	                #sFB_TimerOnOffDelay_Hold330(iudi_OnDelayTime := #cudi_PushOutTime,
	                                             ix_SignalToDelay := NOT #sx_LeftExternalRequestHold330
	                                             AND #iqUDT_WorkstationStatus."310".PEC_EoS.PEC
	                                             AND #iqUDT_WorkstationStatus."320".PEC_EoS.PEC
	                                             AND #iqUDT_WorkstationStatus."330".PEC_EoS.PEC,
	                                             ix_Enable := TRUE);

	                #sFB_TimerOnOffDelay_Hold320(iudi_OnDelayTime := #cudi_PushOutTime,
	                                             ix_SignalToDelay := NOT #sx_LeftExternalRequestHold320
	                                             AND #iqUDT_WorkstationStatus."310".PEC_EoS.PEC
	                                             AND #iqUDT_WorkstationStatus."320".PEC_EoS.PEC,
	                                             ix_Enable := TRUE);

	                #sFB_TimerOnOffDelay_Hold310(iudi_OnDelayTime := #cudi_PushOutTime,
	                                             ix_SignalToDelay := NOT #sx_LeftExternalRequestHold310
	                                             AND #iqUDT_WorkstationStatus."310".PEC_EoS.PEC,
	                                             ix_Enable := TRUE);



	            END_REGION

	            REGION 0.4.2 - Delayed start of pushout conveyors after pushout detection
	                #sFB_TimerOnOffDelay_Detect340(iudi_OnDelayTime := #cudi_DetectTime,
	                                               ix_SignalToDelay := NOT #iqUDT_WorkstationStatus."340".PEC_EoS.PEC,
	                                               ix_Enable := TRUE);

	                #sFB_TimerOnOffDelay_Detect330(iudi_OnDelayTime := #cudi_DetectTime,
	                                               ix_SignalToDelay := NOT #iqUDT_WorkstationStatus."330".PEC_EoS.PEC,
	                                               ix_Enable := TRUE);

	                #sFB_TimerOnOffDelay_Detect320(iudi_OnDelayTime := #cudi_DetectTime,
	                                               ix_SignalToDelay := NOT #iqUDT_WorkstationStatus."320".PEC_EoS.PEC,
	                                               ix_Enable := TRUE);

	                #sFB_TimerOnOffDelay_Detect310(iudi_OnDelayTime := #cudi_DetectTime,
	                                               ix_SignalToDelay := NOT #iqUDT_WorkstationStatus."310".PEC_EoS.PEC,
	                                               ix_Enable := TRUE);
	            END_REGION

	            REGION 0.4.3 - Gate conveyor proximity sensor filtered signal

	                #sFB_TimerOnOffDelay_GateIsDown111Filtered(iudi_OnDelayTime := #cudi_GateIsDownFilterTime,
	                                                           iudi_OffDelayTime := 10,
	                                                           ix_SignalToDelay := #ix_GateIsDown111,
	                                                           qx_DelayedSignal => #sx_GateIsDown111Filtered);
	            END_REGION
	        END_REGION

	        REGION 0.5 - Left station activation

	            IF #sx_ActivationLeft
	            THEN
	                #sx_LeftStationActive := TRUE;
	                #iqUDT_LeftWESInterface.PLC2WES.On := TRUE;
	            END_IF;

	            IF #sx_DeactivationLeft
	            THEN
	                #sx_LeftStationActive := FALSE;
	                #iqUDT_LeftWESInterface.PLC2WES.Off := TRUE;
	            END_IF;


	        END_REGION

	    END_IF;

	END_REGION




	REGION 1 - Initial Right station

	    IF #iUDT_Configuration.GlobalConfig.StationVariant = 1 OR #iUDT_Configuration.GlobalConfig.StationVariant = 3 THEN

	        REGION 1.1 - Reset triggers

	            IF #sx_ActivationRight THEN
	                #iqUDT_RightWESInterface.WES2PLC.On := FALSE;
	                #sx_ActivationRight := FALSE;
	            END_IF;

	            IF #sx_DeactivationRight THEN
	                #iqUDT_RightWESInterface.WES2PLC.Off := FALSE;
	                #sx_DeactivationRight := FALSE;
	            END_IF;

	        END_REGION

	        REGION 1.2 - Triggers

	            #sR_TRIG_PEC540(CLK := #iqUDT_WorkstationStatus."540".PEC_EoS.PEC);   //Rising Edge PEC on conveyor 540 for indexing into station count

	            #sR_TRIG_ActivateRightStation(CLK := #iqUDT_RightWESInterface.WES2PLC.On,     //Rising Edge activate right station
	                                          Q => #sx_ActivationRight);

	            #sR_TRIG_DeactivateRightStation(CLK := #iqUDT_RightWESInterface.WES2PLC.Off,   //Rising Edge deactivate right station
	                                            Q => #sx_DeactivationRight);

	        END_REGION

	        REGION 1.3 - Counters

	            REGION 1.3.1 - Count empty stations on right side

	                //If there is no indexing procedure then count empty stations
	                //
	                IF NOT #sx_RightIndexing THEN

	                    #sFB_CountActiveInputs_RightStation(ix_Input1 := #iqUDT_WorkstationStatus."550".PEC_EoS.PEC,
	                                                        ix_Input2 := #iqUDT_WorkstationStatus."560".PEC_EoS.PEC,
	                                                        ix_Input3 := #iqUDT_WorkstationStatus."570".PEC_EoS.PEC,
	                                                        ix_Input4 := #iqUDT_WorkstationStatus."580".PEC_EoS.PEC,
	                                                        ix_Input5 := #iqUDT_WorkstationStatus."590".PEC_EoS.PEC,
	                                                        qi_ActiveInputsCount => #si_RightEmptyStations);
	                END_IF;
	            END_REGION



	            REGION 1.3.2 - Count free spaces on right buffer

	                IF #sx_RightStationActive THEN
	                    #sFB_CountActiveInputs_RightBuffer(ix_Input1 := #iqUDT_WorkstationStatus."520".PEC_EoS.PEC,
	                                                       ix_Input2 := #iqUDT_WorkstationStatus."530".PEC_EoS.PEC,
	                                                       ix_Input3 := #iqUDT_WorkstationStatus."540".PEC_EoS.PEC);
	                ELSE
	                    #sFB_CountActiveInputs_RightBuffer.qi_ActiveInputsCount := 0;
	                END_IF;

	            END_REGION

	        END_REGION

	        REGION 1.4 - Timers

	            REGION 1.4.1 - Right station timers for holding pushout conveyors after pushout

	                #sFB_TimerOnOffDelay_Hold750(iudi_OnDelayTime := #cudi_PushOutTime,
	                                             ix_SignalToDelay := NOT #sx_RightExternalRequestHold750
	                                             AND #iqUDT_WorkstationStatus."710".PEC_EoS.PEC
	                                             AND #iqUDT_WorkstationStatus."720".PEC_EoS.PEC
	                                             AND #iqUDT_WorkstationStatus."730".PEC_EoS.PEC
	                                             AND #iqUDT_WorkstationStatus."740".PEC_EoS.PEC
	                                             AND #iqUDT_WorkstationStatus."750".PEC_EoS.PEC,
	                                             ix_Enable := TRUE);

	                #sFB_TimerOnOffDelay_Hold740(iudi_OnDelayTime := #cudi_PushOutTime,
	                                             ix_SignalToDelay := NOT #sx_RightExternalRequestHold740
	                                             AND #iqUDT_WorkstationStatus."710".PEC_EoS.PEC
	                                             AND #iqUDT_WorkstationStatus."720".PEC_EoS.PEC
	                                             AND #iqUDT_WorkstationStatus."730".PEC_EoS.PEC
	                                             AND #iqUDT_WorkstationStatus."740".PEC_EoS.PEC,
	                                             ix_Enable := TRUE);

	                #sFB_TimerOnOffDelay_Hold730(iudi_OnDelayTime := #cudi_PushOutTime,
	                                             ix_SignalToDelay := NOT #sx_RightExternalRequestHold730
	                                             AND #iqUDT_WorkstationStatus."710".PEC_EoS.PEC
	                                             AND #iqUDT_WorkstationStatus."720".PEC_EoS.PEC
	                                             AND #iqUDT_WorkstationStatus."730".PEC_EoS.PEC,
	                                             ix_Enable := TRUE);

	                #sFB_TimerOnOffDelay_Hold720(iudi_OnDelayTime := #cudi_PushOutTime,
	                                             ix_SignalToDelay := NOT #sx_RightExternalRequestHold720
	                                             AND #iqUDT_WorkstationStatus."710".PEC_EoS.PEC
	                                             AND #iqUDT_WorkstationStatus."720".PEC_EoS.PEC,
	                                             ix_Enable := TRUE);

	                #sFB_TimerOnOffDelay_Hold710(iudi_OnDelayTime := #cudi_PushOutTime,
	                                             ix_SignalToDelay := NOT #sx_RightExternalRequestHold710
	                                             AND #iqUDT_WorkstationStatus."710".PEC_EoS.PEC,
	                                             ix_Enable := TRUE);
	            END_REGION

	            REGION 1.4.2 - Right station delayed start of pushout conveyors

	                #sFB_TimerOnOffDelay_Detect740(iudi_OnDelayTime := #cudi_DetectTime,
	                                               ix_SignalToDelay := NOT #iqUDT_WorkstationStatus."740".PEC_EoS.PEC,
	                                               ix_Enable := TRUE);

	                #sFB_TimerOnOffDelay_Detect730(iudi_OnDelayTime := #cudi_DetectTime,
	                                               ix_SignalToDelay := NOT #iqUDT_WorkstationStatus."730".PEC_EoS.PEC,
	                                               ix_Enable := TRUE);

	                #sFB_TimerOnOffDelay_Detect720(iudi_OnDelayTime := #cudi_DetectTime,
	                                               ix_SignalToDelay := NOT #iqUDT_WorkstationStatus."720".PEC_EoS.PEC,
	                                               ix_Enable := TRUE);

	                #sFB_TimerOnOffDelay_Detect710(iudi_OnDelayTime := #cudi_DetectTime,
	                                               ix_SignalToDelay := NOT #iqUDT_WorkstationStatus."710".PEC_EoS.PEC,
	                                               ix_Enable := TRUE);

	                #sFB_TimerGateTimeout(iudi_OnDelayTime := #cudi_GateTimout,
	                                      ix_SignalToDelay := NOT #sx_GateIsDown111Filtered,
	                                      qx_DelayedSignal => #sx_GateTimeout);

	            END_REGION

	        END_REGION END_IF;

	        REGION 1.5 - Right station activation

	            IF #sx_ActivationRight
	            THEN
	                #sx_RightStationActive := TRUE;
	                #iqUDT_RightWESInterface.PLC2WES.On := TRUE;
	            END_IF;

	            IF #sx_DeactivationRight
	            THEN
	                #sx_RightStationActive := FALSE;
	                #iqUDT_RightWESInterface.PLC2WES.Off := TRUE;
	            END_IF;

	        END_REGION

	    END_IF;

	END_REGION

	REGION 2 - Lift gate

	    IF #iUDT_Configuration.GlobalConfig.StationVariant > 0 THEN

	        // hold gate conveyors after button press if no maintenance is performed
	        IF #sx_GateIsDown111Filtered AND #sR_TRIG_B112.Q AND NOT #sx_MaintenanceIsPerformed THEN
	            #sx_ExternalRequestHoldGate := TRUE;
	            #sx_MaintenanceIsPerformed := TRUE;


	            // release gate conveyors if gate is down maintenance is performed after button press
	        ELSIF #sx_GateIsDown111Filtered AND #sR_TRIG_B111.Q AND #sx_MaintenanceIsPerformed THEN
	            #sx_ExternalRequestHoldGate := FALSE;
	            #sx_MaintenanceIsPerformed := FALSE;

	            // Hold conveyor if there is no maintenance perfomed and gate has been opened
	        ELSIF NOT #sx_GateIsDown111Filtered AND NOT #sx_MaintenanceIsPerformed THEN
	            #sx_ExternalRequestHoldGate := TRUE;
	        END_IF;


	        // Indicate that Gate is down and stopped
	        IF #sx_MaintenanceIsPerformed AND #sx_GateIsDown111Filtered THEN
	            #qx_Light := TRUE;
	            #sx_HornHold := FALSE;

	            //SCADA Signals
	            #iqUDT_WorkstationStatus."120".LiftGate.Closed := TRUE;
	            #iqUDT_WorkstationStatus."120".LiftGate.Open := FALSE;


	        ELSIF NOT #sx_MaintenanceIsPerformed AND #sx_GateIsDown111Filtered THEN
	            #qx_Light := FALSE;
	            #qx_Horn := FALSE;
	            #sx_HornHold := FALSE;

	        ELSIF NOT #sx_GateIsDown111Filtered AND NOT #sx_GateTimeout THEN
	            #qx_Light := "DB_Memory"."Clock_0.5Hz";

	            IF NOT #sx_HornHold THEN
	                #sx_Horn := TRUE;

	                IF #sx_Horn THEN
	                    #sudi_HornTime += "DB_Memory".PrevCycleTime;
	                    IF #sudi_HornTime > 5000 THEN
	                        #sx_HornHold := TRUE;
	                    END_IF;
	                END_IF;

	            ELSIF #sx_HornHold THEN
	                #sx_Horn := FALSE;
	                #sudi_HornTime := 0;
	            END_IF;
	            #qx_Horn := #sx_Horn;

	            //SCADA Signals
	            #iqUDT_WorkstationStatus."120".LiftGate.Closed := FALSE;
	            #iqUDT_WorkstationStatus."120".LiftGate.Open := TRUE;



	        ELSIF #sx_GateTimeout THEN
	            #qx_Light := "DB_Memory".Clock_2Hz;
	            #qx_Horn := "DB_Memory"."Clock_0.5Hz";
	            #sx_HornHold := FALSE;

	            //SCADA Signals
	            #iqUDT_WorkstationStatus."120".LiftGate.Closed := FALSE;
	            #iqUDT_WorkstationStatus."120".LiftGate.Open := TRUE;
	            #iqUDT_WorkstationStatus."120".LiftGate.Alarms.Timeout := TRUE;


	        END_IF;

	        IF #iqUDT_EquipmentControl.Command.Reset AND #sx_GateIsDown111Filtered THEN   //reset hold and maintenance if gate is closed
	            #sx_ExternalRequestHoldGate := FALSE;
	            #sx_MaintenanceIsPerformed := FALSE;
	            #sx_HornHold := FALSE;

	            //SCADA SIGNALS RESET
	            #iqUDT_WorkstationStatus."120".LiftGate.Closed := FALSE;
	            #iqUDT_WorkstationStatus."120".LiftGate.Open := FALSE;
	            #iqUDT_WorkstationStatus."120".LiftGate.Alarms.Timeout := FALSE;
	        END_IF;


	    END_IF;

	END_REGION

	REGION 3 - Indexing

	    REGION 3.1 - Reset indexing

	        IF #sx_LeftActivateIndex
	        THEN
	            #iqUDT_LeftWESInterface.WES2PLC.Indexing := FALSE;
	            #sx_LeftActivateIndex := FALSE;
	        END_IF;

	        IF #sx_RightActivateIndex
	        THEN
	            #iqUDT_RightWESInterface.WES2PLC.Indexing := FALSE;
	            #sx_RightActivateIndex := FALSE;
	        END_IF;

	        IF #iqUDT_EquipmentControl.Command.Reset
	        THEN
	            #sx_LeftIndexing := FALSE;
	            #sx_RightIndexing := FALSE;
	        END_IF;

	    END_REGION

	    REGION 3.2 - Triggers

	        #sR_TRIG_IndexingLeft(CLK := #iqUDT_LeftWESInterface.WES2PLC.Indexing,
	                              Q => #sx_LeftActivateIndex);


	        #sR_TRIG_IndexingLeft(CLK := #iqUDT_RightWESInterface.WES2PLC.Indexing,
	                              Q => #sx_RightActivateIndex);

	    END_REGION

	END_REGION

	REGION 4 - Middle line
	    REGION Middle RAT divert destinations

	        //Set destination depending on station configuration
	        //If both are configured then divert depending on empty buffer spaces
	        //If buffer spaces count is the same divert to the currently indexed station

	        IF NOT #sx_LeftStationActive AND NOT #sx_RightStationActive THEN
	            #si_DestinationC021 := 0;

	            // ELSIF #sx_LeftStationActive AND NOT #sx_RightStationActive THEN
	            //     // IF #iUDT_Configuration.GlobalConfig.StationVariant = 2 THEN
	            //     #si_DestinationC021 := 2;

	            // ELSIF NOT #sx_LeftStationActive AND #sx_RightStationActive THEN
	            //     //  ELSIF #iUDT_Configuration.GlobalConfig.StationVariant = 3 THEN
	            //     #si_DestinationC021 := 1;

	            // ELSIF #sx_LeftStationActive AND #sx_RightStationActive THEN
	            //  ELSIF #iUDT_Configuration.GlobalConfig.StationVariant = 1 THEN


	        ELSIF #sFB_CountActiveInputs_LeftBuffer.qi_ActiveInputsCount > #sFB_CountActiveInputs_RightBuffer.qi_ActiveInputsCount THEN
	            #si_DestinationC021 := 2;

	        ELSIF #sFB_CountActiveInputs_LeftBuffer.qi_ActiveInputsCount < #sFB_CountActiveInputs_RightBuffer.qi_ActiveInputsCount THEN
	            #si_DestinationC021 := 1;

	        ELSIF #sFB_CountActiveInputs_LeftBuffer.qi_ActiveInputsCount = 0 AND #sFB_CountActiveInputs_RightBuffer.qi_ActiveInputsCount = 0 THEN
	            #si_DestinationC021 := 0;

	        ELSIF #iUDT_Configuration.GlobalConfig.StationVariant = 3 THEN
	            #si_DestinationC021 := 1;

	            // ELSIF #sFB_CountActiveInputs_LeftBuffer.qi_ActiveInputsCount = #sFB_CountActiveInputs_RightBuffer.qi_ActiveInputsCount THEN

	            //     IF #sx_RightIndexing AND NOT #sx_LeftIndexing THEN

	            //         #si_DestinationC021 := 1;

	            //     ELSIF NOT #sx_RightIndexing AND #sx_LeftIndexing THEN

	            //         #si_DestinationC021 := 2;

	            //     ELSIF NOT #sx_RightIndexing AND NOT #sx_LeftIndexing THEN

	            //         #si_DestinationC021 := 1;

	            //   END_IF;
	        END_IF;
	        // END_IF;
	    END_REGION

	    REGION 010

	        REGION Displacement

	            #sFB_Displacement010(#sUDT_Interface010);

	        END_REGION

	        REGION EOS

	            #sFB_PEC010(ix_PEC := #iUDT_MotorInput010.AllSensorPortInputs.LeftSensor,
	                        iUDT_PECConfiguration := #iUDT_Configuration."010".PEC_Eos,
	                        qx_PECFiltered => #tx_dummy,
	                        qUDT_HMIStatus => #iqUDT_WorkstationStatus."010".PEC_EoS,
	                        iqUDT_ConveyorInterface := #sUDT_Interface010,
	                        iqUDT_PECStatistics := #iqUDT_WorkstationStatistics."010".PEC_EoS);

	        END_REGION

	        REGION Conveyor

	            #sUDT_Handshake010.RTR := #sUDT_Handshake010.RTR OR #iqUDT_WorkstationStatus."010".PEC_EoS.PEC;

	            #sFB_Conveyor010(iUDT_ConveyorConfiguration := #iUDT_Configuration."010".Conveyor,
	                             idi_PECEoSDistance := #iUDT_Configuration."010".PEC_Eos.Distance,
	                             idi_PECBoSDistance := 0,
	                             ii_ExternalSpeed := 0,
	                             ix_SafetyOk := #ix_SafetyOk,
	                             ix_24vOk := #ix_24vOk,
	                             ix_400vOk := #ix_400vOk,
	                             ix_HardwareOk := #iUDT_HardwareOk."010",
	                             ix_PECEoS := #iqUDT_WorkstationStatus."010".PEC_EoS.PEC,
	                             ix_PECBoS := TRUE,
	                             ix_ReverseDirection := FALSE,
	                             ix_ExternalRequestDieBack := FALSE,
	                             ix_ExternalRequestHold := FALSE,
	                             ix_ResetEnergySave := FALSE,
	                             qUDT_HMIStatus => #iqUDT_WorkstationStatus."010".Conveyor,
	                             qUDT_Status => #iqUDT_WorkstationCommonStatus."010",
	                             iqUDT_EquipmentControl := #iqUDT_EquipmentControl,
	                             iqUDT_ConveyorCommand := #iqUDT_WorkstationCommands."010".Conveyor,
	                             iqUDT_ConveyorInterface := #sUDT_Interface010,
	                             iqUDT_HandShakeUp := #iqUDT_HandshakeUpstream010,
	                             iqUDT_HandShake := #sUDT_Handshake010,
	                             iqUDT_Statistics := #iqUDT_WorkstationStatistics."010".Conveyor);
	        END_REGION

	        REGION MCO

	            #sFB_MCOConveyLinxAixController010(iUDT_AixConfig := #iUDT_Configuration."010".MCO_M01,
	                                               iv_AixInputsModule := #iUDT_MotorInput010,
	                                               ix_24vOk := #ix_24vOk,
	                                               ix_SimulationModeActive := "DB_Memory".Simulation,
	                                               ii_MotorPositionId := 1,
	                                               qUDT_HMIStatus => #iqUDT_WorkstationStatus."010".MCO_M01,
	                                               iqv_AixOutputsModule := #iqUDT_MotorOutput010,
	                                               iqUDT_ConveyorInterface := #sUDT_Interface010,
	                                               iqUDT_MCOStatistics := #iqUDT_WorkstationStatistics."010".MCO_M01);
	        END_REGION
	    END_REGION

	    REGION 020

	        REGION Displacement

	            #sFB_Displacement020(#sUDT_Interface020);

	        END_REGION

	        REGION MCO

	            #sFB_MCOConveyLinxAixController020(iUDT_AixConfig := #iUDT_Configuration."020".MCO_M01,
	                                               iv_AixInputsModule := #iUDT_MotorInput020,
	                                               ix_24vOk := #ix_24vOk,
	                                               ix_SimulationModeActive := "DB_Memory".Simulation,
	                                               ii_MotorPositionId := 1,
	                                               qUDT_HMIStatus => #iqUDT_WorkstationStatus."020".MCO_M01,
	                                               iqv_AixOutputsModule := #iqUDT_MotorOutput020,
	                                               iqUDT_ConveyorInterface := #sUDT_Interface020,
	                                               iqUDT_MCOStatistics := #iqUDT_WorkstationStatistics."020".MCO_M01);
	        END_REGION
	    END_REGION

	    REGION 021

	        REGION Displacement

	            #sFB_Displacement021(#sUDT_Interface021);

	        END_REGION

	        REGION RAT

	            IF #iUDT_Configuration.GlobalConfig.StationVariant = 1 OR #iUDT_Configuration.GlobalConfig.StationVariant = 2 THEN
	                #sUDT_Handshake021B := #sUDT_Handshake110A;
	                #sUDT_Handshake021A := #sUDT_Handshake510A;
	            ELSIF #iUDT_Configuration.GlobalConfig.StationVariant = 3 THEN
	                #sUDT_Handshake021A := #sUDT_Handshake110A;
	            END_IF;



	            #sFB_RightAngledTransfer021(iUDT_Configuration := #iUDT_Configuration."021".RightAngledTransfer,
	                                        iUDT_LowerConveyorConfiguration := #iUDT_Configuration."020".Conveyor,
	                                        iUDT_UpperConveyorConfiguration := #iUDT_Configuration."021".Conveyor,
	                                        iUDT_PECConfiguration := #iUDT_Configuration."020".PEC_EoS,
	                                        ii_DestinationA := 0,
	                                        ii_DestinationB := 0,
	                                        ii_DestinationC := #si_DestinationC021,
	                                        ii_DestinationD := 0,
	                                        ix_HardwareOk := #iUDT_HardwareOk."020",
	                                        ix_400vOk := #ix_400vOk,
	                                        ix_24vOk := #ix_24vOk,
	                                        ix_SafetyOk := #ix_SafetyOk,
	                                        ix_AirPressureOk := #ix_AirPressureOk,
	                                        ix_SectionIsDown := #ix_SectionIsDown021,
	                                        ix_SectionIsUp := #ix_SectionIsUp021,
	                                        ix_ConveyorAAuto := FALSE,
	                                        ix_ConveyorBAuto := false,
	                                        ix_ConveyorCAuto := #iqUDT_WorkstationCommonStatus."010".AutoON,
	                                        ix_ConveyorDAuto := false,
	                                        ix_PEC := #iUDT_MotorInput020.AllSensorPortInputs.LeftSensor,
	                                        ix_ExternalReceiveRequestA := FALSE,
	                                        ix_ExternalReceiveRequestB := FALSE,
	                                        ix_ExternalReceiveRequestC := NOT #iqUDT_WorkstationStatus."010".PEC_EoS.PEC,
	                                        ix_ExternalReceiveRequestD := FALSE,
	                                        ix_PECInfeedC := #iqUDT_WorkstationStatus."010".PEC_EoS.PEC,
	                                        qUDT_HMIRATStatus => #iqUDT_WorkstationStatus."021".RightAngledTransfer,
	                                        qUDT_HMIConveyorStatus => #iqUDT_WorkstationStatus."020".Conveyor,
	                                        qUDT_HMIPECStatus => #iqUDT_WorkstationStatus."020".PEC_EoS,
	                                        qUDT_RATStatus => #iqUDT_WorkstationCommonStatus."021",
	                                        qUDT_ConveyorStatus => #iqUDT_WorkstationCommonStatus."020",
	                                        qx_PopupControl => #qx_PopupControl021,
	                                        qx_ExternalSendRequestA => #tx_dummy,
	                                        qx_ExternalSendRequestB => #tx_dummy,
	                                        qx_ExternalSendRequestC => #tx_dummy,
	                                        qx_ExternalSendRequestD => #tx_dummy,
	                                        iqUDT_EquipmentControl := #iqUDT_EquipmentControl,
	                                        iqUDT_RATCommand := #iqUDT_WorkstationCommands."021".RightAngledTransfer,
	                                        iqUDT_ConveyorCommand := #iqUDT_WorkstationCommands."020".Conveyor,
	                                        iqUDT_RATStatistics := #iqUDT_WorkstationStatistics."021".RightAngledTransfer,
	                                        iqUDT_ConveyorStatistics := #iqUDT_WorkstationStatistics."020".Conveyor,
	                                        iqUDT_PECStatistics := #iqUDT_WorkstationStatistics."020".PEC_EoS,
	                                        iqUDT_HandShakeConveyorA := #sUDT_Handshake021A,
	                                        iqUDT_HandShakeConveyorB := #sUDT_Handshake021B,
	                                        iqUDT_HandShakeConveyorC := #sUDT_Handshake010,
	                                        iqUDT_HandShakeConveyorD := #tUDT_DummyConveyorHandshake,
	                                        iqUDT_LowerConveyorInterface := #sUDT_Interface020,
	                                        iqUDT_UpperConveyorInterface := #sUDT_Interface021,
	                                        iqUDT_RATPositioning := #iqUDT_RATPositioning020,
	                                        iqUDT_BladeStopEoSInterface := #tUDT_DummyBladeStop,
	                                        iqUDT_BladeStopBoSInterface := #tUDT_DummyBladeStop);

	        END_REGION


	        IF #iUDT_Configuration.GlobalConfig.StationVariant = 1 OR #iUDT_Configuration.GlobalConfig.StationVariant = 2 THEN
	            #sUDT_Handshake110A := #sUDT_Handshake021B;
	            #sUDT_Handshake510A := #sUDT_Handshake021A;
	        ELSIF #iUDT_Configuration.GlobalConfig.StationVariant = 3 THEN
	            #sUDT_Handshake110A := #sUDT_Handshake021A;
	        END_IF;

	        REGION MCO

	            #sFB_MCOConveyLinxAixController021(iUDT_AixConfig := #iUDT_Configuration."021".MCO_M01,
	                                               iv_AixInputsModule := #iUDT_MotorInput020,
	                                               ii_PositionSetpoint := #iqUDT_RATPositioning020.Upper.EndPosition,
	                                               ix_24vOk := #ix_24vOk,
	                                               ix_SimulationModeActive := "DB_Memory".Simulation,
	                                               ii_MotorPositionId := 2,
	                                               ix_StartPositioning := #iqUDT_RATPositioning020.Upper.Start,
	                                               ix_ResetPosition := #iqUDT_RATPositioning020.Upper.ResetPosition,
	                                               qUDT_HMIStatus => #iqUDT_WorkstationStatus."021".MCO_M01,
	                                               qx_Positioned => #iqUDT_RATPositioning020.Upper.Done,
	                                               iqv_AixOutputsModule := #iqUDT_MotorOutput020,
	                                               iqUDT_ConveyorInterface := #sUDT_Interface021,
	                                               iqUDT_MCOStatistics := #iqUDT_WorkstationStatistics."021".MCO_M01);
	        END_REGION

	    END_REGION

	END_REGION

	REGION 5 - Left Station

	    IF #iUDT_Configuration.GlobalConfig.StationVariant > 0 THEN

	        REGION 5.1 - Indexing

	            // Start indexing after request if there are empty stations and no pushout is active

	            IF #sx_LeftActivateIndex AND #si_LeftEmptyStations > 0
	                AND NOT (#sx_LeftPushOutActiveStation1
	                OR #sx_LeftPushOutActiveStation2
	                OR #sx_LeftPushOutActiveStation3
	                OR #sx_LeftPushOutActiveStation4
	                OR #sx_LeftPushOutActiveStation5) THEN

	                #sx_LeftIndexing := TRUE;

	            END_IF;

	            IF NOT #sx_LeftIndexing THEN                           // If there is no indexing in progress

	                #si_LeftDestinationC141 := 0;                     // Reset RAT destination
	                #sx_LeftExternalRequestHold150 := TRUE;           // Hold station conveyors
	                #sx_LeftExternalRequestHold160 := TRUE;
	                #sx_LeftExternalRequestHold170 := TRUE;
	                #sx_LeftExternalRequestHold180 := TRUE;
	                #sx_LeftExternalRequestHold190 := TRUE;

	            ELSE                                                // If there is indexing in progress

	                IF #sR_TRIG_PEC140.Q AND #si_LeftEmptyStations > 0 THEN  //Count down empty stations after diverting a tote into station
	                    #si_LeftEmptyStations -= 1;
	                END_IF;

	                IF #iUDT_Configuration.GlobalConfig.StationVariant = 3 THEN
	                    #si_LeftDestinationC141 := 4;
	                ELSE
	                    #si_LeftDestinationC141 := 3;
	                END_IF;

	                #sx_LeftExternalRequestHold150 := FALSE;           // Release hold of station conveyors and set RAT destination
	                #sx_LeftExternalRequestHold160 := FALSE;
	                #sx_LeftExternalRequestHold170 := FALSE;
	                #sx_LeftExternalRequestHold180 := FALSE;
	                #sx_LeftExternalRequestHold190 := FALSE;

	                IF
	                    NOT #iqUDT_WorkstationStatus."150".PEC_EoS.PEC       //End indexing when all totes are on position
	                    AND NOT #iqUDT_WorkstationStatus."160".PEC_EoS.PEC
	                    AND NOT #iqUDT_WorkstationStatus."170".PEC_EoS.PEC
	                    AND NOT #iqUDT_WorkstationStatus."180".PEC_EoS.PEC
	                    AND NOT #iqUDT_WorkstationStatus."190".PEC_EoS.PEC
	                    AND NOT (#sUDT_Interface150.ActualSpeed > 0) THEN

	                    #sx_LeftIndexing := FALSE;

	                END_IF;

	            END_IF;

	        END_REGION

	        REGION 5.2 - Push Out

	            IF #iUDT_Configuration.GlobalConfig.LeftCubbyNumbering = 1 THEN
	                #sa_LeftCubby[1] := 10;
	                #sa_LeftCubby[2] := 9;
	                #sa_LeftCubby[3] := 8;
	                #sa_LeftCubby[4] := 7;
	                #sa_LeftCubby[5] := 6;
	            ELSIF #iUDT_Configuration.GlobalConfig.LeftCubbyNumbering = 2 THEN
	                #sa_LeftCubby[1] := 5;
	                #sa_LeftCubby[2] := 4;
	                #sa_LeftCubby[3] := 3;
	                #sa_LeftCubby[4] := 2;
	                #sa_LeftCubby[5] := 1;
	            END_IF;

	            IF #iUDT_Configuration.GlobalConfig.StationVariant = 3 THEN
	                IF #iUDT_Configuration.GlobalConfig.RightCubbyNumbering = 1 THEN
	                    #sa_LeftCubby[1] := 10;
	                    #sa_LeftCubby[2] := 9;
	                    #sa_LeftCubby[3] := 8;
	                    #sa_LeftCubby[4] := 7;
	                    #sa_LeftCubby[5] := 6;
	                ELSIF #iUDT_Configuration.GlobalConfig.RightCubbyNumbering = 2 THEN
	                    #sa_LeftCubby[1] := 5;
	                    #sa_LeftCubby[2] := 4;
	                    #sa_LeftCubby[3] := 3;
	                    #sa_LeftCubby[4] := 2;
	                    #sa_LeftCubby[5] := 1;
	                END_IF;
	            END_IF;

	            REGION 5.2.0 Pushout conveyors hold

	                IF #sFB_TimerOnOffDelay_Hold310.qx_DelayedSignal THEN
	                    #sx_LeftExternalRequestHold310 := TRUE;
	                END_IF;

	                IF #sFB_TimerOnOffDelay_Hold320.qx_DelayedSignal THEN
	                    #sx_LeftExternalRequestHold320 := TRUE;
	                END_IF;

	                IF #sFB_TimerOnOffDelay_Hold330.qx_DelayedSignal THEN
	                    #sx_LeftExternalRequestHold330 := TRUE;
	                END_IF;

	                IF #sFB_TimerOnOffDelay_Hold340.qx_DelayedSignal THEN
	                    #sx_LeftExternalRequestHold340 := TRUE;
	                END_IF;

	                IF #sFB_TimerOnOffDelay_Hold350.qx_DelayedSignal THEN
	                    #sx_LeftExternalRequestHold350 := TRUE;
	                END_IF;
	            END_REGION

	            REGION 5.2.1 - Push Out Station 1



	                // Start automatic pushout after request if there is no indexing procedure and a tote is present on first station
	                IF #iqUDT_LeftWESInterface.Field[#sa_LeftCubby[1]].WES2PLC.RemoveContainer AND NOT #sx_LeftIndexing
	                    AND NOT #iqUDT_WorkstationStatus."190".PEC_EoS.PEC THEN

	                    #sx_LeftPushOutActiveStation1 := TRUE;
	                    #iqUDT_LeftWESInterface.Field[#sa_LeftCubby[1]].WES2PLC.RemoveContainer := FALSE;
	                END_IF;

	                IF #sx_LeftPushOutActiveStation1 THEN
	                    #sx_LeftExternalRequestHold190 := FALSE;    //release hold

	                    IF #sFB_RightAngledTransfer211.qx_ExternalSendRequestB THEN   //after tote is already on RAT, hold the conveyor and end pushout procedure
	                        #sx_LeftExternalRequestHold190 := TRUE;
	                        #sx_LeftPushOutActiveStation1 := FALSE;
	                    END_IF;
	                END_IF;

	            END_REGION

	            REGION 5.2.2 - Push Out station 2

	                IF #iqUDT_LeftWESInterface.Field[#sa_LeftCubby[2]].WES2PLC.RemoveContainer THEN //set pushout to active after request
	                    #sx_LeftPushOutActiveStation2 := TRUE;
	                    #iqUDT_LeftWESInterface.Field[#sa_LeftCubby[2]].WES2PLC.RemoveContainer := FALSE;
	                END_IF;

	                IF #sx_LeftPushOutActiveStation2              // After station is empty and tote has been detected on pushout conveyor release holds
	                    AND #iqUDT_WorkstationStatus."180".PEC_EoS.PEC
	                    AND #sFB_TimerOnOffDelay_Detect340.qx_DelayedSignal THEN

	                    #sx_LeftExternalRequestHold340 := FALSE;
	                    #sx_LeftExternalRequestHold350 := FALSE;

	                    FILL_BLK(IN := 0,                                 //clear tracking
	                             COUNT := REAL_TO_ULINT(DINT_TO_REAL(#iUDT_Configuration."180".Conveyor.Common.Length) * #cr_ClearTrackingModifier),
	                             OUT => #sa_TrackingArray180[0]);

	                    #sx_LeftPushOutActiveStation2 := FALSE;            //end pushout procedure

	                END_IF;


	            END_REGION

	            REGION 5.2.3 - Push Out station 3

	                IF #iqUDT_LeftWESInterface.Field[#sa_LeftCubby[3]].WES2PLC.RemoveContainer THEN        //set pushout to active after request
	                    #sx_LeftPushOutActiveStation3 := TRUE;
	                    #iqUDT_LeftWESInterface.Field[#sa_LeftCubby[3]].WES2PLC.RemoveContainer := FALSE;
	                END_IF;

	                IF #sx_LeftPushOutActiveStation3                             // After station is empty and tote has been detected on pushout conveyor release holds
	                    AND #iqUDT_WorkstationStatus."170".PEC_EoS.PEC
	                    AND #sFB_TimerOnOffDelay_Detect330.qx_DelayedSignal THEN

	                    #sx_LeftExternalRequestHold330 := FALSE;
	                    #sx_LeftExternalRequestHold340 := FALSE;
	                    #sx_LeftExternalRequestHold350 := FALSE;

	                    FILL_BLK(IN := 0,                                      //clear tracking
	                             COUNT := REAL_TO_ULINT(DINT_TO_REAL(#iUDT_Configuration."170".Conveyor.Common.Length) * #cr_ClearTrackingModifier),
	                             OUT => #sa_TrackingArray170[0]);

	                    #sx_LeftPushOutActiveStation3 := FALSE;                  //end pushout procedure

	                END_IF;
	            END_REGION

	            REGION 5.2.4 - Push Out station 4

	                IF #iqUDT_LeftWESInterface.Field[#sa_LeftCubby[4]].WES2PLC.RemoveContainer THEN         //set pushout to active after request
	                    #sx_LeftPushOutActiveStation4 := TRUE;
	                    #iqUDT_LeftWESInterface.Field[#sa_LeftCubby[4]].WES2PLC.RemoveContainer := FALSE;
	                END_IF;

	                IF #sx_LeftPushOutActiveStation4                           // After station is empty and tote has been detected on pushout conveyor release holds
	                    AND #iqUDT_WorkstationStatus."160".PEC_EoS.PEC
	                    AND #sFB_TimerOnOffDelay_Detect320.qx_DelayedSignal THEN

	                    #sx_LeftExternalRequestHold320 := FALSE;
	                    #sx_LeftExternalRequestHold330 := FALSE;
	                    #sx_LeftExternalRequestHold340 := FALSE;
	                    #sx_LeftExternalRequestHold350 := FALSE;

	                    FILL_BLK(IN := 0,                                     //clear tracking
	                             COUNT := REAL_TO_ULINT(DINT_TO_REAL(#iUDT_Configuration."160".Conveyor.Common.Length) * #cr_ClearTrackingModifier),
	                             OUT => #sa_TrackingArray160[0]);

	                    #sx_LeftPushOutActiveStation4 := FALSE;               //end pushout procedure

	                END_IF;

	            END_REGION

	            REGION 5.2.5 - Push Out station 5

	                IF #iqUDT_LeftWESInterface.Field[#sa_LeftCubby[5]].WES2PLC.RemoveContainer THEN          //set pushout to active after request
	                    #sx_LeftPushOutActiveStation5 := TRUE;
	                    #iqUDT_LeftWESInterface.Field[#sa_LeftCubby[5]].WES2PLC.RemoveContainer := FALSE;
	                END_IF;

	                IF #sx_LeftPushOutActiveStation5                                   // After station is empty and tote has been detected on pushout conveyor release holds
	                    AND #iqUDT_WorkstationStatus."150".PEC_EoS.PEC
	                    AND #sFB_TimerOnOffDelay_Detect310.qx_DelayedSignal THEN

	                    #sx_LeftExternalRequestHold310 := FALSE;
	                    #sx_LeftExternalRequestHold320 := FALSE;
	                    #sx_LeftExternalRequestHold330 := FALSE;
	                    #sx_LeftExternalRequestHold340 := FALSE;
	                    #sx_LeftExternalRequestHold350 := FALSE;

	                    FILL_BLK(IN := 0,                                                 //clear tracking
	                             COUNT := REAL_TO_ULINT(DINT_TO_REAL(#iUDT_Configuration."150".Conveyor.Common.Length) * #cr_ClearTrackingModifier),
	                             OUT => #sa_TrackingArray150[0]);

	                    #sx_LeftPushOutActiveStation5 := FALSE;                     //end pushout procedure
	                END_IF;

	            END_REGION

	            REGION 5.2.6 - Pushout support logic
	                IF #iUDT_Configuration.GlobalConfig.PushoutsPresent AND
	                    ((#iUDT_Configuration.GlobalConfig.StationVariant = 1 OR
	                    #iUDT_Configuration.GlobalConfig.StationVariant = 2)) THEN

	                    IF (NOT #iqUDT_WorkstationStatus."150".PEC_EoS.PEC AND #sx_LeftPushOutActiveStation5) OR
	                        (NOT #iqUDT_WorkstationStatus."160".PEC_EoS.PEC AND #sx_LeftPushOutActiveStation4) THEN
	                        #sx_Hold360 := FALSE;

	                    ELSIF NOT (#sx_LeftPushOutActiveStation4 OR #sx_LeftPushOutActiveStation5) THEN
	                        #sx_Hold360 := TRUE; //Hold pushout conveyors

	                    END_IF;

	                    //Package present on the left side pecs, pushouts run
	                    IF (NOT #iqUDT_WorkstationStatus."170".PEC_EoS.PEC AND #sx_LeftPushOutActiveStation3) OR
	                        (#sx_LeftPushOutActiveStation2 AND NOT #iqUDT_WorkstationStatus."180".PEC_EoS.PEC) THEN
	                        #sx_Hold370 := FALSE;

	                    ELSIF NOT (#sx_LeftPushOutActiveStation3 OR #sx_LeftPushOutActiveStation2) THEN
	                        #sx_Hold370 := TRUE; //Hold pushout conveyors

	                    END_IF;
	                END_IF;
	            END_REGION



	        END_REGION

	        REGION 5.3 WES communication

	            REGION 5.3.2 Barcode to WES
	                IF NOT #sx_LeftIndexing
	                THEN

	                    REGION 190
	                        // first position
	                        //
	                        IF NOT #sx_LeftPushOutActiveStation1
	                            AND NOT #iqUDT_WorkstationStatus."190".PEC_EoS.PEC
	                            AND #sa_TrackingArray190[(#iUDT_Configuration."190".PEC_Eos.Distance / 10) - 1] > 0
	                        THEN

	                            IF #iqUDT_LeftWESInterface.Field[#sa_LeftCubby[1]].WES2PLC.SetContainerID THEN

	                                "DB_GIN".GIN[#sa_TrackingArray190[(#iUDT_Configuration."190".PEC_Eos.Distance / 10) - 1]].General.Identification.Barcode := #iqUDT_LeftWESInterface.Field[#sa_LeftCubby[1]].WES2PLC.ContainerID;
	                                #iqUDT_LeftWESInterface.Field[#sa_LeftCubby[1]].WES2PLC.SetContainerID := FALSE;

	                            END_IF;

	                            IF #iqUDT_LeftWESInterface.Field[#sa_LeftCubby[1]].PLC2WES.ContainerID <> "DB_GIN".GIN[#sa_TrackingArray190[(#iUDT_Configuration."190".PEC_Eos.Distance / 10) - 1]].General.Identification.Barcode
	                            THEN

	                                #iqUDT_LeftWESInterface.Field[#sa_LeftCubby[1]].PLC2WES.ContainerID := "DB_GIN".GIN[#sa_TrackingArray190[(#iUDT_Configuration."190".PEC_Eos.Distance / 10) - 1]].General.Identification.Barcode;
	                                #iqUDT_LeftWESInterface.Field[#sa_LeftCubby[1]].PLC2WES.SetContainerID := TRUE;
	                            END_IF;

	                        ELSE
	                            IF #iqUDT_LeftWESInterface.Field[#sa_LeftCubby[1]].PLC2WES.ContainerID <> #cs_MissingBarcodeCode
	                            THEN
	                                #iqUDT_LeftWESInterface.Field[#sa_LeftCubby[1]].PLC2WES.ContainerID := #cs_MissingBarcodeCode;
	                                #iqUDT_LeftWESInterface.Field[#sa_LeftCubby[1]].PLC2WES.SetContainerID := TRUE;

	                            END_IF;

	                        END_IF;
	                    END_REGION ;
	                    REGION 180
	                        // second position
	                        //
	                        IF NOT #iqUDT_WorkstationStatus."180".PEC_EoS.PEC
	                            AND #sa_TrackingArray180[(#iUDT_Configuration."180".PEC_Eos.Distance / 10) - 1] > 0
	                        THEN

	                            IF #iqUDT_LeftWESInterface.Field[#sa_LeftCubby[2]].WES2PLC.SetContainerID THEN

	                                "DB_GIN".GIN[#sa_TrackingArray180[(#iUDT_Configuration."180".PEC_Eos.Distance / 10) - 1]].General.Identification.Barcode := #iqUDT_LeftWESInterface.Field[#sa_LeftCubby[2]].WES2PLC.ContainerID;
	                                #iqUDT_LeftWESInterface.Field[#sa_LeftCubby[2]].WES2PLC.SetContainerID := FALSE;

	                            END_IF;

	                            IF #iqUDT_LeftWESInterface.Field[#sa_LeftCubby[2]].PLC2WES.ContainerID <> "DB_GIN".GIN[#sa_TrackingArray180[(#iUDT_Configuration."180".PEC_Eos.Distance / 10) - 1]].General.Identification.Barcode
	                            THEN

	                                #iqUDT_LeftWESInterface.Field[#sa_LeftCubby[2]].PLC2WES.ContainerID := "DB_GIN".GIN[#sa_TrackingArray180[(#iUDT_Configuration."180".PEC_Eos.Distance / 10) - 1]].General.Identification.Barcode;
	                                #iqUDT_LeftWESInterface.Field[#sa_LeftCubby[2]].PLC2WES.SetContainerID := TRUE;
	                            END_IF;

	                        ELSE
	                            IF #iqUDT_LeftWESInterface.Field[#sa_LeftCubby[2]].PLC2WES.ContainerID <> #cs_MissingBarcodeCode
	                            THEN
	                                #iqUDT_LeftWESInterface.Field[#sa_LeftCubby[2]].PLC2WES.ContainerID := #cs_MissingBarcodeCode;
	                                #iqUDT_LeftWESInterface.Field[#sa_LeftCubby[2]].PLC2WES.SetContainerID := TRUE;

	                            END_IF;

	                        END_IF;
	                    END_REGION ;
	                    REGION 170
	                        // third position
	                        //
	                        IF NOT #iqUDT_WorkstationStatus."170".PEC_EoS.PEC
	                            AND #sa_TrackingArray170[(#iUDT_Configuration."170".PEC_Eos.Distance / 10) - 1] > 0
	                        THEN

	                            IF #iqUDT_LeftWESInterface.Field[#sa_LeftCubby[3]].WES2PLC.SetContainerID THEN

	                                "DB_GIN".GIN[#sa_TrackingArray170[(#iUDT_Configuration."170".PEC_Eos.Distance / 10) - 1]].General.Identification.Barcode := #iqUDT_LeftWESInterface.Field[#sa_LeftCubby[3]].WES2PLC.ContainerID;
	                                #iqUDT_LeftWESInterface.Field[#sa_LeftCubby[3]].WES2PLC.SetContainerID := FALSE;

	                            END_IF;

	                            IF #iqUDT_LeftWESInterface.Field[#sa_LeftCubby[3]].PLC2WES.ContainerID <> "DB_GIN".GIN[#sa_TrackingArray170[(#iUDT_Configuration."170".PEC_Eos.Distance / 10) - 1]].General.Identification.Barcode
	                            THEN

	                                #iqUDT_LeftWESInterface.Field[#sa_LeftCubby[3]].PLC2WES.ContainerID := "DB_GIN".GIN[#sa_TrackingArray170[(#iUDT_Configuration."170".PEC_Eos.Distance / 10) - 1]].General.Identification.Barcode;
	                                #iqUDT_LeftWESInterface.Field[#sa_LeftCubby[3]].PLC2WES.SetContainerID := TRUE;
	                            END_IF;

	                        ELSE
	                            IF #iqUDT_LeftWESInterface.Field[#sa_LeftCubby[3]].PLC2WES.ContainerID <> #cs_MissingBarcodeCode
	                            THEN
	                                #iqUDT_LeftWESInterface.Field[#sa_LeftCubby[3]].PLC2WES.ContainerID := #cs_MissingBarcodeCode;
	                                #iqUDT_LeftWESInterface.Field[#sa_LeftCubby[3]].PLC2WES.SetContainerID := TRUE;

	                            END_IF;

	                        END_IF;
	                    END_REGION ;
	                    REGION 160
	                        // fourth position
	                        //
	                        IF NOT #iqUDT_WorkstationStatus."160".PEC_EoS.PEC
	                            AND #sa_TrackingArray160[(#iUDT_Configuration."160".PEC_Eos.Distance / 10) - 1] > 0
	                        THEN

	                            IF #iqUDT_LeftWESInterface.Field[#sa_LeftCubby[4]].WES2PLC.SetContainerID THEN

	                                "DB_GIN".GIN[#sa_TrackingArray160[(#iUDT_Configuration."160".PEC_Eos.Distance / 10) - 1]].General.Identification.Barcode := #iqUDT_LeftWESInterface.Field[#sa_LeftCubby[4]].WES2PLC.ContainerID;
	                                #iqUDT_LeftWESInterface.Field[#sa_LeftCubby[4]].WES2PLC.SetContainerID := FALSE;

	                            END_IF;

	                            IF #iqUDT_LeftWESInterface.Field[#sa_LeftCubby[4]].PLC2WES.ContainerID <> "DB_GIN".GIN[#sa_TrackingArray160[(#iUDT_Configuration."160".PEC_Eos.Distance / 10) - 1]].General.Identification.Barcode
	                            THEN

	                                #iqUDT_LeftWESInterface.Field[#sa_LeftCubby[4]].PLC2WES.ContainerID := "DB_GIN".GIN[#sa_TrackingArray160[(#iUDT_Configuration."160".PEC_Eos.Distance / 10) - 1]].General.Identification.Barcode;
	                                #iqUDT_LeftWESInterface.Field[#sa_LeftCubby[4]].PLC2WES.SetContainerID := TRUE;
	                            END_IF;

	                        ELSE
	                            IF #iqUDT_LeftWESInterface.Field[#sa_LeftCubby[4]].PLC2WES.ContainerID <> #cs_MissingBarcodeCode
	                            THEN
	                                #iqUDT_LeftWESInterface.Field[#sa_LeftCubby[4]].PLC2WES.ContainerID := #cs_MissingBarcodeCode;
	                                #iqUDT_LeftWESInterface.Field[#sa_LeftCubby[4]].PLC2WES.SetContainerID := TRUE;

	                            END_IF;

	                        END_IF;
	                    END_REGION ;
	                    REGION 150
	                        //fifth position
	                        //
	                        IF NOT #iqUDT_WorkstationStatus."150".PEC_EoS.PEC
	                            AND #sa_TrackingArray150[(#iUDT_Configuration."150".PEC_Eos.Distance / 10) - 1] > 0
	                        THEN

	                            IF #iqUDT_LeftWESInterface.Field[#sa_LeftCubby[5]].WES2PLC.SetContainerID THEN

	                                "DB_GIN".GIN[#sa_TrackingArray150[(#iUDT_Configuration."150".PEC_Eos.Distance / 10) - 1]].General.Identification.Barcode := #iqUDT_LeftWESInterface.Field[#sa_LeftCubby[5]].WES2PLC.ContainerID;
	                                #iqUDT_LeftWESInterface.Field[#sa_LeftCubby[5]].WES2PLC.SetContainerID := FALSE;

	                            END_IF;

	                            IF #iqUDT_LeftWESInterface.Field[#sa_LeftCubby[5]].PLC2WES.ContainerID <> "DB_GIN".GIN[#sa_TrackingArray150[(#iUDT_Configuration."150".PEC_Eos.Distance / 10) - 1]].General.Identification.Barcode
	                            THEN

	                                #iqUDT_LeftWESInterface.Field[#sa_LeftCubby[5]].PLC2WES.ContainerID := "DB_GIN".GIN[#sa_TrackingArray150[(#iUDT_Configuration."150".PEC_Eos.Distance / 10) - 1]].General.Identification.Barcode;
	                                #iqUDT_LeftWESInterface.Field[#sa_LeftCubby[5]].PLC2WES.SetContainerID := TRUE;
	                            END_IF;

	                        ELSE
	                            IF #iqUDT_LeftWESInterface.Field[#sa_LeftCubby[5]].PLC2WES.ContainerID <> #cs_MissingBarcodeCode
	                            THEN
	                                #iqUDT_LeftWESInterface.Field[#sa_LeftCubby[5]].PLC2WES.ContainerID := #cs_MissingBarcodeCode;
	                                #iqUDT_LeftWESInterface.Field[#sa_LeftCubby[5]].PLC2WES.SetContainerID := TRUE;

	                            END_IF;

	                        END_IF;
	                    END_REGION ;

	                END_IF;


	            END_REGION

	        END_REGION

	        REGION 5.4 Function Block calls

	            REGION 110

	                REGION Displacement

	                    #sFB_Displacement110(#sUDT_Interface110);

	                END_REGION

	                REGION Tracking
	                    #sFB_Tracking110(iUDT_ConveyorCommonConfiguration := #iUDT_Configuration."110".Conveyor.Common,
	                                     iqa_TrackingData := #sa_TrackingArray110,
	                                     iqUDT_ConveyorInterface := #sUDT_Interface110,
	                                     iqUDT_HandshakeUp := #sUDT_Handshake020,
	                                     iqUDT_Handshake := #sUDT_Handshake110);

	                END_REGION

	                REGION EOS
	                    #sFB_PECUpdate110(iUDT_PECUpdateConfiguration := #iUDT_Configuration."110".PEC_Eos,
	                                      iUDT_ConveyorCommonConfiguration := #iUDT_Configuration."110".Conveyor.Common,
	                                      ix_PEC := NOT #iUDT_MotorInput110.AllSensorPortInputs.LeftSensor,
	                                      ix_TeachingMode := FALSE,
	                                      qUDT_Status => #iqUDT_WorkstationStatus."110".PEC_EoS,
	                                      qi_GINwrite => #ti_dummy,
	                                      qx_PECFiltered => #tx_dummy,
	                                      iqUDT_ConveyorInterface := #sUDT_Interface110,
	                                      iqUDT_UnknownGINRange := #iqUDT_UnknownGINRange,
	                                      iqUDT_FifoHeader := "DB_FIFOLostGIN".Header,
	                                      iqUDT_Statistics := #iqUDT_WorkstationStatistics."110".PEC_EoS,
	                                      iqa_TrackingData := #sa_TrackingArray110,
	                                      iqa_FifoData := "DB_FIFOLostGIN".Data);

	                END_REGION

	                REGION Conveyor

	                    #sFB_Conveyor110(iUDT_ConveyorConfiguration := #iUDT_Configuration."110".Conveyor,
	                                     idi_PECEoSDistance := #iUDT_Configuration."110".PEC_Eos.Distance,
	                                     idi_PECBoSDistance := 0,
	                                     ii_ExternalSpeed := 0,
	                                     ix_SafetyOk := #ix_SafetyOk,
	                                     ix_24vOk := #ix_24vOk,
	                                     ix_400vOk := #ix_400vOk,
	                                     ix_HardwareOk := #iUDT_HardwareOk."110",
	                                     ix_PECEoS := #iqUDT_WorkstationStatus."110".PEC_EoS.PEC,
	                                     ix_PECBoS := TRUE,
	                                     ix_ReverseDirection := FALSE,
	                                     ix_ExternalRequestDieBack := FALSE,
	                                     ix_ExternalRequestHold := (NOT #sx_GateIsDown111Filtered OR #sx_ExternalRequestHoldGate),
	                                     ix_ResetEnergySave := FALSE,
	                                     qUDT_HMIStatus => #iqUDT_WorkstationStatus."110".Conveyor,
	                                     qUDT_Status => #iqUDT_WorkstationCommonStatus."110",
	                                     iqUDT_EquipmentControl := #iqUDT_EquipmentControl,
	                                     iqUDT_ConveyorCommand := #iqUDT_WorkstationCommands."110".Conveyor,
	                                     iqUDT_ConveyorInterface := #sUDT_Interface110,
	                                     iqUDT_HandShakeUp := #sUDT_Handshake110A,
	                                     iqUDT_HandShake := #sUDT_Handshake110,
	                                     iqUDT_Statistics := #iqUDT_WorkstationStatistics."110".Conveyor);

	                END_REGION

	                REGION MCO

	                    #sFB_MCOConveyLinxAixController110(iUDT_AixConfig := #iUDT_Configuration."110".MCO_M01,
	                                                       iv_AixInputsModule := #iUDT_MotorInput110,
	                                                       ix_24vOk := #ix_24vOk,
	                                                       ix_SimulationModeActive := "DB_Memory".Simulation,
	                                                       ii_MotorPositionId := 1,
	                                                       qUDT_HMIStatus => #iqUDT_WorkstationStatus."110".MCO_M01,
	                                                       iqv_AixOutputsModule := #iqUDT_MotorOutput110,
	                                                       iqUDT_ConveyorInterface := #sUDT_Interface110,
	                                                       iqUDT_MCOStatistics := #iqUDT_WorkstationStatistics."110".MCO_M01);
	                END_REGION
	            END_REGION

	            REGION 120

	                REGION Displacement

	                    #sFB_Displacement120(#sUDT_Interface120);

	                END_REGION

	                REGION Tracking

	                    #sFB_Tracking120(iUDT_ConveyorCommonConfiguration := #iUDT_Configuration."120".Conveyor.Common,
	                                     iqa_TrackingData := #sa_TrackingArray120,
	                                     iqUDT_ConveyorInterface := #sUDT_Interface120,
	                                     iqUDT_HandshakeUp := #sUDT_Handshake110,
	                                     iqUDT_Handshake := #sUDT_Handshake120);

	                END_REGION

	                REGION Conveyor

	                    #sFB_Conveyor120(iUDT_ConveyorConfiguration := #iUDT_Configuration."120".Conveyor,
	                                     idi_PECEoSDistance := 0,
	                                     idi_PECBoSDistance := 0,
	                                     ii_ExternalSpeed := 0,
	                                     ix_SafetyOk := #ix_SafetyOk,
	                                     ix_24vOk := #ix_24vOk,
	                                     ix_400vOk := #ix_400vOk,
	                                     ix_HardwareOk := #iUDT_HardwareOk."110",
	                                     ix_PECEoS := TRUE,
	                                     ix_PECBoS := TRUE,
	                                     ix_ReverseDirection := FALSE,
	                                     ix_ExternalRequestDieBack := FALSE,
	                                     ix_ExternalRequestHold := (NOT #sx_GateIsDown111Filtered OR #sx_ExternalRequestHoldGate),
	                                     ix_ResetEnergySave := FALSE,
	                                     qUDT_HMIStatus => #iqUDT_WorkstationStatus."120".Conveyor,
	                                     qUDT_Status => #iqUDT_WorkstationCommonStatus."120",
	                                     iqUDT_EquipmentControl := #iqUDT_EquipmentControl,
	                                     iqUDT_ConveyorCommand := #iqUDT_WorkstationCommands."120".Conveyor,
	                                     iqUDT_ConveyorInterface := #sUDT_Interface120,
	                                     iqUDT_HandShakeUp := #sUDT_Handshake110,
	                                     iqUDT_HandShake := #sUDT_Handshake120,
	                                     iqUDT_Statistics := #iqUDT_WorkstationStatistics."120".Conveyor);
	                END_REGION

	                REGION MCO

	                    #sFB_MCOConveyLinxAixController120(iUDT_AixConfig := #iUDT_Configuration."120".MCO_M01,
	                                                       iv_AixInputsModule := #iUDT_MotorInput110,
	                                                       ix_24vOk := #ix_24vOk,
	                                                       ix_SimulationModeActive := "DB_Memory".Simulation,
	                                                       ii_MotorPositionId := 2,
	                                                       qUDT_HMIStatus => #iqUDT_WorkstationStatus."120".MCO_M01,
	                                                       iqv_AixOutputsModule := #iqUDT_MotorOutput110,
	                                                       iqUDT_ConveyorInterface := #sUDT_Interface120,
	                                                       iqUDT_MCOStatistics := #iqUDT_WorkstationStatistics."120".MCO_M01);
	                END_REGION

	            END_REGION

	            REGION 130

	                REGION Displacement

	                    #sFB_Displacement130(#sUDT_Interface130);

	                END_REGION

	                REGION Tracking

	                    #sFB_Tracking130(iUDT_ConveyorCommonConfiguration := #iUDT_Configuration."130".Conveyor.Common,
	                                     iqa_TrackingData := #sa_TrackingArray130,
	                                     iqUDT_ConveyorInterface := #sUDT_Interface130,
	                                     iqUDT_HandshakeUp := #sUDT_Handshake120,
	                                     iqUDT_Handshake := #sUDT_Handshake130);

	                END_REGION

	                REGION EOS
	                    #sFB_PECUpdate130(iUDT_PECUpdateConfiguration := #iUDT_Configuration."130".PEC_Eos,
	                                      iUDT_ConveyorCommonConfiguration := #iUDT_Configuration."130".Conveyor.Common,
	                                      ix_PEC := NOT #iUDT_MotorInput130.AllSensorPortInputs.LeftSensor,
	                                      ix_TeachingMode := FALSE,
	                                      qUDT_Status => #iqUDT_WorkstationStatus."130".PEC_EoS,
	                                      qi_GINwrite => #ti_dummy,
	                                      qx_PECFiltered => #tx_dummy,
	                                      iqUDT_ConveyorInterface := #sUDT_Interface130,
	                                      iqUDT_UnknownGINRange := #iqUDT_UnknownGINRange,
	                                      iqUDT_FifoHeader := "DB_FIFOLostGIN".Header,
	                                      iqUDT_Statistics := #iqUDT_WorkstationStatistics."130".PEC_EoS,
	                                      iqa_TrackingData := #sa_TrackingArray130,
	                                      iqa_FifoData := "DB_FIFOLostGIN".Data);

	                END_REGION



	                REGION Conveyor

	                    //  #sUDT_Handshake130.RTR := #iqUDT_WorkstationStatus."130".PEC_EoS.PEC OR
	                    // (#iqUDT_WorkstationStatus."140".PEC_EoS.PEC AND #sUDT_Interface140.ActualSpeed <> 0);

	                    #sFB_Conveyor130(iUDT_ConveyorConfiguration := #iUDT_Configuration."130".Conveyor,
	                                     idi_PECEoSDistance := #iUDT_Configuration."130".PEC_Eos.Distance,
	                                     idi_PECBoSDistance := 0,
	                                     ii_ExternalSpeed := 0,
	                                     ix_SafetyOk := #ix_SafetyOk,
	                                     ix_24vOk := #ix_24vOk,
	                                     ix_400vOk := #ix_400vOk,
	                                     ix_HardwareOk := #iUDT_HardwareOk."130",
	                                     ix_PECEoS := #iqUDT_WorkstationStatus."130".PEC_EoS.PEC,
	                                     ix_PECBoS := TRUE,
	                                     ix_ReverseDirection := FALSE,
	                                     ix_ExternalRequestDieBack := FALSE,
	                                     ix_ExternalRequestHold := FALSE,
	                                     ix_ResetEnergySave := FALSE,
	                                     qUDT_HMIStatus => #iqUDT_WorkstationStatus."130".Conveyor,
	                                     qUDT_Status => #iqUDT_WorkstationCommonStatus."130",
	                                     iqUDT_EquipmentControl := #iqUDT_EquipmentControl,
	                                     iqUDT_ConveyorCommand := #iqUDT_WorkstationCommands."130".Conveyor,
	                                     iqUDT_ConveyorInterface := #sUDT_Interface130,
	                                     iqUDT_HandShakeUp := #sUDT_Handshake120,
	                                     iqUDT_HandShake := #sUDT_Handshake130,
	                                     iqUDT_Statistics := #iqUDT_WorkstationStatistics."130".Conveyor);
	                END_REGION

	                REGION MCO

	                    #sFB_MCOConveyLinxAixController130(iUDT_AixConfig := #iUDT_Configuration."130".MCO_M01,
	                                                       iv_AixInputsModule := #iUDT_MotorInput130,
	                                                       ix_24vOk := #ix_24vOk,
	                                                       ix_SimulationModeActive := "DB_Memory".Simulation,
	                                                       ii_MotorPositionId := 1,
	                                                       qUDT_HMIStatus => #iqUDT_WorkstationStatus."130".MCO_M01,
	                                                       iqv_AixOutputsModule := #iqUDT_MotorOutput130,
	                                                       iqUDT_ConveyorInterface := #sUDT_Interface130,
	                                                       iqUDT_MCOStatistics := #iqUDT_WorkstationStatistics."130".MCO_M01);
	                END_REGION
	            END_REGION

	            REGION 131
	                REGION Scanner

	                    #sFB_DataLogicBlade131(iUDT_ScannerInput := #iUDT_ScannerInput131,
	                                           iUDT_ScannerConfiguration := #iUDT_Configuration."131".Scanner,
	                                           iUDT_ConveyorInterface := #sUDT_Interface130,
	                                           ii_GIN := #sa_TrackingArray130[#iUDT_Configuration."131".Scanner.ScannerPosition],
	                                           ix_24vOk := #ix_24vOk,
	                                           ix_HardwareOk := #iUDT_HardwareOk."131",
	                                           ix_SimulationModeActive := "DB_Memory".Simulation,
	                                           qUDT_ScannerOutput => #qUDT_ScannerOutput131,
	                                           qUDT_HMIStatus => #iqUDT_WorkstationStatus."131".Scanner,
	                                           qUDT_CommonStatus => #iqUDT_WorkstationCommonStatus."131",
	                                           iqUDT_Statistics := #iqUDT_WorkstationStatistics."131".Scanner,
	                                           iqUDT_EquipmentControl := #iqUDT_EquipmentControl);


	                END_REGION
	            END_REGION

	            REGION 140

	                REGION Displacement

	                    #sFB_Displacement140(#sUDT_Interface140);

	                END_REGION

	                REGION MCO

	                    #sFB_MCOConveyLinxAixController140(iUDT_AixConfig := #iUDT_Configuration."140".MCO_M01,
	                                                       iv_AixInputsModule := #iUDT_MotorInput140,
	                                                       ii_PositionSetpoint := #iqUDT_RATPositioning140.Lower.EndPosition,
	                                                       ix_24vOk := #ix_24vOk,
	                                                       ix_SimulationModeActive := "DB_Memory".Simulation,
	                                                       ii_MotorPositionId := 1,
	                                                       ix_StartPositioning := #iqUDT_RATPositioning140.Lower.Start,
	                                                       ix_ResetPosition := #iqUDT_RATPositioning140.Lower.ResetPosition,
	                                                       qUDT_HMIStatus => #iqUDT_WorkstationStatus."140".MCO_M01,
	                                                       qx_Positioned => #iqUDT_RATPositioning140.Lower.Done,
	                                                       iqv_AixOutputsModule := #iqUDT_MotorOutput140,
	                                                       iqUDT_ConveyorInterface := #sUDT_Interface140,
	                                                       iqUDT_MCOStatistics := #iqUDT_WorkstationStatistics."140".MCO_M01);
	                END_REGION
	            END_REGION

	            REGION 141

	                REGION Displacement

	                    #sFB_Displacement141(#sUDT_Interface141);

	                END_REGION

	                REGION RAT

	                    #sUDT_Handshake141.RTR := #sx_LeftIndexing AND
	                    (#iqUDT_WorkstationStatus."150".PEC_EoS.PEC AND #sUDT_Interface150.ActualSpeed <> 0);

	                    IF #iUDT_Configuration.GlobalConfig.StationVariant = 1 OR #iUDT_Configuration.GlobalConfig.StationVariant = 2 THEN
	                        #sUDT_Handshake141C := #sUDT_Handshake141;
	                    ELSIF #iUDT_Configuration.GlobalConfig.StationVariant = 3 THEN
	                        #sUDT_Handshake141D := #sUDT_Handshake141;
	                    END_IF;





	                    #sFB_RightAngledTransfer141(iUDT_Configuration := #iUDT_Configuration."141".RightAngledTransfer,
	                                                iUDT_LowerConveyorConfiguration := #iUDT_Configuration."140".Conveyor,
	                                                iUDT_UpperConveyorConfiguration := #iUDT_Configuration."141".Conveyor,
	                                                iUDT_PECConfiguration := #iUDT_Configuration."140".PEC_EoS,
	                                                ii_DestinationA := #si_LeftDestinationC141,
	                                                ii_DestinationB := 0,
	                                                ii_DestinationC := 0,
	                                                ii_DestinationD := 0,
	                                                ix_HardwareOk := #iUDT_HardwareOk."140",
	                                                ix_400vOk := #ix_400vOk,
	                                                ix_24vOk := #ix_24vOk,
	                                                ix_SafetyOk := #ix_SafetyOk,
	                                                ix_AirPressureOk := #ix_AirPressureOk,
	                                                ix_SectionIsDown := #ix_SectionIsDown141,
	                                                ix_SectionIsUp := #ix_SectionIsUp141,
	                                                ix_ConveyorAAuto := #iqUDT_WorkstationCommonStatus."130".AutoON,
	                                                ix_ConveyorBAuto := false,
	                                                ix_ConveyorCAuto := false,
	                                                ix_ConveyorDAuto := false,
	                                                ix_PEC := #iUDT_MotorInput140.AllSensorPortInputs.LeftSensor,
	                                                ix_ExternalReceiveRequestA := NOT #iqUDT_WorkstationStatus."130".PEC_EoS.PEC,
	                                                ix_ExternalReceiveRequestB := FALSE,
	                                                ix_ExternalReceiveRequestC := FALSE,
	                                                ix_ExternalReceiveRequestD := FALSE,
	                                                ix_PECInfeedA := #iqUDT_WorkstationStatus."130".PEC_EoS.PEC,
	                                                qUDT_HMIRATStatus => #iqUDT_WorkstationStatus."141".RightAngledTransfer,
	                                                qUDT_HMIConveyorStatus => #iqUDT_WorkstationStatus."140".Conveyor,
	                                                qUDT_HMIPECStatus => #iqUDT_WorkstationStatus."140".PEC_EoS,
	                                                qUDT_RATStatus => #iqUDT_WorkstationCommonStatus."141",
	                                                qUDT_ConveyorStatus => #iqUDT_WorkstationCommonStatus."140",
	                                                qx_PopupControl => #qx_PopupControl141,
	                                                qx_ExternalSendRequestA => #tx_dummy,
	                                                qx_ExternalSendRequestB => #tx_dummy,
	                                                qx_ExternalSendRequestC => #tx_dummy,
	                                                qx_ExternalSendRequestD => #tx_dummy,
	                                                iqUDT_EquipmentControl := #iqUDT_EquipmentControl,
	                                                iqUDT_RATCommand := #iqUDT_WorkstationCommands."141".RightAngledTransfer,
	                                                iqUDT_ConveyorCommand := #iqUDT_WorkstationCommands."140".Conveyor,
	                                                iqUDT_RATStatistics := #iqUDT_WorkstationStatistics."141".RightAngledTransfer,
	                                                iqUDT_ConveyorStatistics := #iqUDT_WorkstationStatistics."140".Conveyor,
	                                                iqUDT_PECStatistics := #iqUDT_WorkstationStatistics."140".PEC_EoS,
	                                                iqUDT_HandShakeConveyorA := #sUDT_Handshake130,
	                                                iqUDT_HandShakeConveyorB := #tUDT_DummyConveyorHandshake,
	                                                iqUDT_HandShakeConveyorC := #sUDT_Handshake141C,
	                                                iqUDT_HandShakeConveyorD := #sUDT_Handshake141D,
	                                                iqUDT_LowerConveyorInterface := #sUDT_Interface140,
	                                                iqUDT_UpperConveyorInterface := #sUDT_Interface141,
	                                                iqUDT_RATPositioning := #iqUDT_RATPositioning140,
	                                                iqUDT_BladeStopEoSInterface := #tUDT_DummyBladeStop,
	                                                iqUDT_BladeStopBoSInterface := #tUDT_DummyBladeStop);

	                END_REGION

	                IF #iUDT_Configuration.GlobalConfig.StationVariant = 1 OR #iUDT_Configuration.GlobalConfig.StationVariant = 2 THEN
	                    #sUDT_Handshake141 := #sUDT_Handshake141C;
	                ELSIF #iUDT_Configuration.GlobalConfig.StationVariant = 3 THEN
	                    #sUDT_Handshake141 := #sUDT_Handshake141D;
	                END_IF;


	                REGION MCO

	                    #sFB_MCOConveyLinxAixController141(iUDT_AixConfig := #iUDT_Configuration."141".MCO_M01,
	                                                       iv_AixInputsModule := #iUDT_MotorInput140,
	                                                       ix_24vOk := #ix_24vOk,
	                                                       ix_SimulationModeActive := "DB_Memory".Simulation,
	                                                       ii_MotorPositionId := 2,
	                                                       qUDT_HMIStatus => #iqUDT_WorkstationStatus."141".MCO_M01,
	                                                       iqv_AixOutputsModule := #iqUDT_MotorOutput140,
	                                                       iqUDT_ConveyorInterface := #sUDT_Interface141,
	                                                       iqUDT_MCOStatistics := #iqUDT_WorkstationStatistics."141".MCO_M01);
	                END_REGION

	            END_REGION

	            REGION 150

	                REGION Displacement

	                    #sFB_Displacement150(#sUDT_Interface150);

	                END_REGION

	                REGION Tracking

	                    #sFB_Tracking150(iUDT_ConveyorCommonConfiguration := #iUDT_Configuration."150".Conveyor.Common,
	                                     iqa_TrackingData := #sa_TrackingArray150,
	                                     iqUDT_ConveyorInterface := #sUDT_Interface150,
	                                     iqUDT_HandshakeUp := #sUDT_Handshake141,
	                                     iqUDT_Handshake := #sUDT_Handshake150);
	                END_REGION

	                REGION EOS

	                    #sFB_PECUpdate150(iUDT_PECUpdateConfiguration := #iUDT_Configuration."150".PEC_Eos,
	                                      iUDT_ConveyorCommonConfiguration := #iUDT_Configuration."150".Conveyor.Common,
	                                      ix_PEC := NOT #iUDT_MotorInput150.AllSensorPortInputs.LeftSensor,
	                                      ix_TeachingMode := FALSE,
	                                      qUDT_Status => #iqUDT_WorkstationStatus."150".PEC_EoS,
	                                      qi_GINwrite => #ti_dummy,
	                                      qx_PECFiltered => #tx_dummy,
	                                      iqa_TrackingData := #sa_TrackingArray150,
	                                      iqUDT_ConveyorInterface := #sUDT_Interface150,
	                                      iqUDT_UnknownGINRange := #iqUDT_UnknownGINRange,
	                                      iqUDT_FifoHeader := "DB_FIFOLostGIN".Header,
	                                      iqa_FifoData := "DB_FIFOLostGIN".Data,
	                                      iqUDT_Statistics := #iqUDT_WorkstationStatistics."150".PEC_EoS);

	                END_REGION

	                REGION Conveyor

	                    #sUDT_Handshake150.RTR := #sx_LeftIndexing AND
	                    ((#iqUDT_WorkstationStatus."160".PEC_EoS.PEC AND #sUDT_Interface160.ActualSpeed <> 0) OR #iqUDT_WorkstationStatus."150".PEC_EoS.PEC);

	                    #sFB_Conveyor150(iUDT_ConveyorConfiguration := #iUDT_Configuration."150".Conveyor,
	                                     idi_PECEoSDistance := #iUDT_Configuration."150".PEC_Eos.Distance,
	                                     idi_PECBoSDistance := 0,
	                                     ii_ExternalSpeed := 0,
	                                     ix_SafetyOk := #ix_SafetyOk,
	                                     ix_24vOk := #ix_24vOk,
	                                     ix_400vOk := #ix_400vOk,
	                                     ix_HardwareOk := #iUDT_HardwareOk."150",
	                                     ix_PECEoS := #iqUDT_WorkstationStatus."150".PEC_EoS.PEC,
	                                     ix_PECBoS := TRUE,
	                                     ix_ReverseDirection := FALSE,
	                                     ix_ExternalRequestDieBack := FALSE,
	                                     ix_ExternalRequestHold := #sx_LeftExternalRequestHold150,
	                                     ix_ResetEnergySave := FALSE,
	                                     qUDT_HMIStatus => #iqUDT_WorkstationStatus."150".Conveyor,
	                                     qUDT_Status => #iqUDT_WorkstationCommonStatus."150",
	                                     iqUDT_EquipmentControl := #iqUDT_EquipmentControl,
	                                     iqUDT_ConveyorCommand := #iqUDT_WorkstationCommands."150".Conveyor,
	                                     iqUDT_ConveyorInterface := #sUDT_Interface150,
	                                     iqUDT_HandShakeUp := #sUDT_Handshake141,
	                                     iqUDT_HandShake := #sUDT_Handshake150,
	                                     iqUDT_Statistics := #iqUDT_WorkstationStatistics."150".Conveyor);
	                END_REGION

	                REGION MCO

	                    #sFB_MCOConveyLinxAixController150(iUDT_AixConfig := #iUDT_Configuration."150".MCO_M01,
	                                                       iv_AixInputsModule := #iUDT_MotorInput150,
	                                                       ix_24vOk := #ix_24vOk,
	                                                       ix_SimulationModeActive := "DB_Memory".Simulation,
	                                                       ii_MotorPositionId := 1,
	                                                       qUDT_HMIStatus => #iqUDT_WorkstationStatus."150".MCO_M01,
	                                                       iqv_AixOutputsModule := #iqUDT_MotorOutput150,
	                                                       iqUDT_ConveyorInterface := #sUDT_Interface150,
	                                                       iqUDT_MCOStatistics := #iqUDT_WorkstationStatistics."150".MCO_M01);
	                END_REGION

	            END_REGION

	            REGION 160

	                REGION Displacement

	                    #sFB_Displacement160(#sUDT_Interface160);

	                END_REGION

	                REGION Tracking

	                    #sFB_Tracking160(iUDT_ConveyorCommonConfiguration := #iUDT_Configuration."160".Conveyor.Common,
	                                     iqa_TrackingData := #sa_TrackingArray160,
	                                     iqUDT_ConveyorInterface := #sUDT_Interface160,
	                                     iqUDT_HandshakeUp := #sUDT_Handshake150,
	                                     iqUDT_Handshake := #sUDT_Handshake160);
	                END_REGION

	                REGION EOS

	                    #sFB_PECUpdate160(iUDT_PECUpdateConfiguration := #iUDT_Configuration."160".PEC_Eos,
	                                      iUDT_ConveyorCommonConfiguration := #iUDT_Configuration."160".Conveyor.Common,
	                                      ix_PEC := NOT #iUDT_MotorInput150.AllSensorPortInputs.RightSensor,
	                                      ix_TeachingMode := FALSE,
	                                      qUDT_Status => #iqUDT_WorkstationStatus."160".PEC_EoS,
	                                      qi_GINwrite => #ti_dummy,
	                                      qx_PECFiltered => #tx_dummy,
	                                      iqa_TrackingData := #sa_TrackingArray160,
	                                      iqUDT_ConveyorInterface := #sUDT_Interface160,
	                                      iqUDT_UnknownGINRange := #iqUDT_UnknownGINRange,
	                                      iqUDT_FifoHeader := "DB_FIFOLostGIN".Header,
	                                      iqa_FifoData := "DB_FIFOLostGIN".Data,
	                                      iqUDT_Statistics := #iqUDT_WorkstationStatistics."160".PEC_EoS);

	                END_REGION

	                REGION Conveyor

	                    #sUDT_Handshake160.RTR := #sx_LeftIndexing AND
	                    ((#iqUDT_WorkstationStatus."170".PEC_EoS.PEC AND #sUDT_Interface170.ActualSpeed <> 0) OR #iqUDT_WorkstationStatus."160".PEC_EoS.PEC);

	                    #sFB_Conveyor160(iUDT_ConveyorConfiguration := #iUDT_Configuration."160".Conveyor,
	                                     idi_PECEoSDistance := #iUDT_Configuration."160".PEC_Eos.Distance,
	                                     idi_PECBoSDistance := 0,
	                                     ii_ExternalSpeed := 0,
	                                     ix_SafetyOk := #ix_SafetyOk,
	                                     ix_24vOk := #ix_24vOk,
	                                     ix_400vOk := #ix_400vOk,
	                                     ix_HardwareOk := #iUDT_HardwareOk."150",
	                                     ix_PECEoS := #iqUDT_WorkstationStatus."160".PEC_EoS.PEC,
	                                     ix_PECBoS := TRUE,
	                                     ix_ReverseDirection := FALSE,
	                                     ix_ExternalRequestDieBack := FALSE,
	                                     ix_ExternalRequestHold := #sx_LeftExternalRequestHold160,
	                                     ix_ResetEnergySave := FALSE,
	                                     qUDT_HMIStatus => #iqUDT_WorkstationStatus."160".Conveyor,
	                                     qUDT_Status => #iqUDT_WorkstationCommonStatus."160",
	                                     iqUDT_EquipmentControl := #iqUDT_EquipmentControl,
	                                     iqUDT_ConveyorCommand := #iqUDT_WorkstationCommands."160".Conveyor,
	                                     iqUDT_ConveyorInterface := #sUDT_Interface160,
	                                     iqUDT_HandShakeUp := #sUDT_Handshake150,
	                                     iqUDT_HandShake := #sUDT_Handshake160,
	                                     iqUDT_Statistics := #iqUDT_WorkstationStatistics."160".Conveyor);
	                END_REGION

	                REGION MCO

	                    #sFB_MCOConveyLinxAixController160(iUDT_AixConfig := #iUDT_Configuration."160".MCO_M01,
	                                                       iv_AixInputsModule := #iUDT_MotorInput150,
	                                                       ix_24vOk := #ix_24vOk,
	                                                       ix_SimulationModeActive := "DB_Memory".Simulation,
	                                                       ii_MotorPositionId := 2,
	                                                       qUDT_HMIStatus => #iqUDT_WorkstationStatus."160".MCO_M01,
	                                                       iqv_AixOutputsModule := #iqUDT_MotorOutput150,
	                                                       iqUDT_ConveyorInterface := #sUDT_Interface160,
	                                                       iqUDT_MCOStatistics := #iqUDT_WorkstationStatistics."160".MCO_M01);
	                END_REGION
	            END_REGION

	            REGION 170

	                REGION Displacement

	                    #sFB_Displacement170(#sUDT_Interface170);

	                END_REGION

	                REGION Tracking

	                    #sFB_Tracking170(iUDT_ConveyorCommonConfiguration := #iUDT_Configuration."170".Conveyor.Common,
	                                     iqa_TrackingData := #sa_TrackingArray170,
	                                     iqUDT_ConveyorInterface := #sUDT_Interface170,
	                                     iqUDT_HandshakeUp := #sUDT_Handshake160,
	                                     iqUDT_Handshake := #sUDT_Handshake170);
	                END_REGION

	                REGION EOS

	                    #sFB_PECUpdate170(iUDT_PECUpdateConfiguration := #iUDT_Configuration."170".PEC_Eos,
	                                      iUDT_ConveyorCommonConfiguration := #iUDT_Configuration."170".Conveyor.Common,
	                                      ix_PEC := NOT #iUDT_MotorInput170.AllSensorPortInputs.LeftSensor,
	                                      ix_TeachingMode := FALSE,
	                                      qUDT_Status => #iqUDT_WorkstationStatus."170".PEC_EoS,
	                                      qi_GINwrite => #ti_dummy,
	                                      qx_PECFiltered => #tx_dummy,
	                                      iqa_TrackingData := #sa_TrackingArray170,
	                                      iqUDT_ConveyorInterface := #sUDT_Interface170,
	                                      iqUDT_UnknownGINRange := #iqUDT_UnknownGINRange,
	                                      iqUDT_FifoHeader := "DB_FIFOLostGIN".Header,
	                                      iqa_FifoData := "DB_FIFOLostGIN".Data,
	                                      iqUDT_Statistics := #iqUDT_WorkstationStatistics."170".PEC_EoS);

	                END_REGION

	                REGION Conveyor

	                    #sUDT_Handshake170.RTR := #sx_LeftIndexing AND
	                    ((#iqUDT_WorkstationStatus."180".PEC_EoS.PEC AND #sUDT_Interface180.ActualSpeed <> 0) OR #iqUDT_WorkstationStatus."170".PEC_EoS.PEC);

	                    #sFB_Conveyor170(iUDT_ConveyorConfiguration := #iUDT_Configuration."170".Conveyor,
	                                     idi_PECEoSDistance := #iUDT_Configuration."170".PEC_Eos.Distance,
	                                     idi_PECBoSDistance := 0,
	                                     ii_ExternalSpeed := 0,
	                                     ix_SafetyOk := #ix_SafetyOk,
	                                     ix_24vOk := #ix_24vOk,
	                                     ix_400vOk := #ix_400vOk,
	                                     ix_HardwareOk := #iUDT_HardwareOk."170",
	                                     ix_PECEoS := #iqUDT_WorkstationStatus."170".PEC_EoS.PEC,
	                                     ix_PECBoS := TRUE,
	                                     ix_ExternalRequestHold := #sx_LeftExternalRequestHold170,
	                                     qUDT_HMIStatus => #iqUDT_WorkstationStatus."170".Conveyor,
	                                     qUDT_Status => #iqUDT_WorkstationCommonStatus."170",
	                                     iqUDT_EquipmentControl := #iqUDT_EquipmentControl,
	                                     iqUDT_ConveyorCommand := #iqUDT_WorkstationCommands."170".Conveyor,
	                                     iqUDT_ConveyorInterface := #sUDT_Interface170,
	                                     iqUDT_HandShakeUp := #sUDT_Handshake160,
	                                     iqUDT_HandShake := #sUDT_Handshake170,
	                                     iqUDT_Statistics := #iqUDT_WorkstationStatistics."170".Conveyor);
	                END_REGION

	                REGION MCO

	                    #sFB_MCOConveyLinxAixController170(iUDT_AixConfig := #iUDT_Configuration."170".MCO_M01,
	                                                       iv_AixInputsModule := #iUDT_MotorInput170,
	                                                       ix_24vOk := #ix_24vOk,
	                                                       ix_SimulationModeActive := "DB_Memory".Simulation,
	                                                       ii_MotorPositionId := 1,
	                                                       qUDT_HMIStatus => #iqUDT_WorkstationStatus."170".MCO_M01,
	                                                       iqv_AixOutputsModule := #iqUDT_MotorOutput170,
	                                                       iqUDT_ConveyorInterface := #sUDT_Interface170,
	                                                       iqUDT_MCOStatistics := #iqUDT_WorkstationStatistics."170".MCO_M01);
	                END_REGION
	            END_REGION

	            REGION 180

	                REGION Displacement

	                    #sFB_Displacement180(#sUDT_Interface180);

	                END_REGION

	                REGION Tracking

	                    #sFB_Tracking180(iUDT_ConveyorCommonConfiguration := #iUDT_Configuration."180".Conveyor.Common,
	                                     iqa_TrackingData := #sa_TrackingArray180,
	                                     iqUDT_ConveyorInterface := #sUDT_Interface180,
	                                     iqUDT_HandshakeUp := #sUDT_Handshake170,
	                                     iqUDT_Handshake := #sUDT_Handshake180);
	                END_REGION

	                REGION EOS

	                    #sFB_PECUpdate180(iUDT_PECUpdateConfiguration := #iUDT_Configuration."180".PEC_Eos,
	                                      iUDT_ConveyorCommonConfiguration := #iUDT_Configuration."180".Conveyor.Common,
	                                      ix_PEC := NOT #iUDT_MotorInput170.AllSensorPortInputs.RightSensor,
	                                      ix_TeachingMode := FALSE,
	                                      qUDT_Status => #iqUDT_WorkstationStatus."180".PEC_EoS,
	                                      qi_GINwrite => #ti_dummy,
	                                      qx_PECFiltered => #tx_dummy,
	                                      iqa_TrackingData := #sa_TrackingArray180,
	                                      iqUDT_ConveyorInterface := #sUDT_Interface180,
	                                      iqUDT_UnknownGINRange := #iqUDT_UnknownGINRange,
	                                      iqUDT_FifoHeader := "DB_FIFOLostGIN".Header,
	                                      iqa_FifoData := "DB_FIFOLostGIN".Data,
	                                      iqUDT_Statistics := #iqUDT_WorkstationStatistics."180".PEC_EoS);

	                END_REGION

	                REGION Conveyor

	                    #sUDT_Handshake180.RTR := #sx_LeftIndexing AND
	                    ((#iqUDT_WorkstationStatus."190".PEC_EoS.PEC AND #sUDT_Interface190.ActualSpeed <> 0) OR #iqUDT_WorkstationStatus."180".PEC_EoS.PEC);

	                    #sFB_Conveyor180(iUDT_ConveyorConfiguration := #iUDT_Configuration."180".Conveyor,
	                                     idi_PECEoSDistance := #iUDT_Configuration."180".PEC_Eos.Distance,
	                                     idi_PECBoSDistance := 0,
	                                     ii_ExternalSpeed := 0,
	                                     ix_SafetyOk := #ix_SafetyOk,
	                                     ix_24vOk := #ix_24vOk,
	                                     ix_400vOk := #ix_400vOk,
	                                     ix_HardwareOk := #iUDT_HardwareOk."170",
	                                     ix_PECEoS := #iqUDT_WorkstationStatus."180".PEC_EoS.PEC,
	                                     ix_PECBoS := TRUE,
	                                     ix_ReverseDirection := FALSE,
	                                     ix_ExternalRequestDieBack := FALSE,
	                                     ix_ExternalRequestHold := #sx_LeftExternalRequestHold180,
	                                     ix_ResetEnergySave := FALSE,
	                                     qUDT_HMIStatus => #iqUDT_WorkstationStatus."180".Conveyor,
	                                     qUDT_Status => #iqUDT_WorkstationCommonStatus."180",
	                                     iqUDT_EquipmentControl := #iqUDT_EquipmentControl,
	                                     iqUDT_ConveyorCommand := #iqUDT_WorkstationCommands."180".Conveyor,
	                                     iqUDT_ConveyorInterface := #sUDT_Interface180,
	                                     iqUDT_HandShakeUp := #sUDT_Handshake170,
	                                     iqUDT_HandShake := #sUDT_Handshake180,
	                                     iqUDT_Statistics := #iqUDT_WorkstationStatistics."180".Conveyor);
	                END_REGION

	                REGION MCO

	                    #sFB_MCOConveyLinxAixController180(iUDT_AixConfig := #iUDT_Configuration."180".MCO_M01,
	                                                       iv_AixInputsModule := #iUDT_MotorInput170,
	                                                       ix_24vOk := #ix_24vOk,
	                                                       ix_SimulationModeActive := "DB_Memory".Simulation,
	                                                       ii_MotorPositionId := 2,
	                                                       qUDT_HMIStatus => #iqUDT_WorkstationStatus."180".MCO_M01,
	                                                       iqv_AixOutputsModule := #iqUDT_MotorOutput170,
	                                                       iqUDT_ConveyorInterface := #sUDT_Interface180,
	                                                       iqUDT_MCOStatistics := #iqUDT_WorkstationStatistics."180".MCO_M01);
	                END_REGION

	            END_REGION

	            REGION 190

	                REGION Displacement

	                    #sFB_Displacement190(#sUDT_Interface190);

	                END_REGION

	                REGION Tracking

	                    #sFB_Tracking190(iUDT_ConveyorCommonConfiguration := #iUDT_Configuration."190".Conveyor.Common,
	                                     iqa_TrackingData := #sa_TrackingArray190,
	                                     iqUDT_ConveyorInterface := #sUDT_Interface190,
	                                     iqUDT_HandshakeUp := #sUDT_Handshake180,
	                                     iqUDT_Handshake := #sUDT_Handshake190);
	                END_REGION

	                REGION EOS

	                    #sFB_PECUpdate190(iUDT_PECUpdateConfiguration := #iUDT_Configuration."190".PEC_Eos,
	                                      iUDT_ConveyorCommonConfiguration := #iUDT_Configuration."190".Conveyor.Common,
	                                      ix_PEC := NOT #iUDT_MotorInput190.AllSensorPortInputs.LeftSensor,
	                                      ix_TeachingMode := FALSE,
	                                      qUDT_Status => #iqUDT_WorkstationStatus."190".PEC_EoS,
	                                      qi_GINwrite => #ti_dummy,
	                                      qx_PECFiltered => #tx_dummy,
	                                      iqa_TrackingData := #sa_TrackingArray190,
	                                      iqUDT_ConveyorInterface := #sUDT_Interface190,
	                                      iqUDT_UnknownGINRange := #iqUDT_UnknownGINRange,
	                                      iqUDT_FifoHeader := "DB_FIFOLostGIN".Header,
	                                      iqa_FifoData := "DB_FIFOLostGIN".Data,
	                                      iqUDT_Statistics := #iqUDT_WorkstationStatistics."190".PEC_EoS);

	                END_REGION

	                REGION Conveyor

	                    #sUDT_Handshake190.RTR := (#sx_LeftIndexing AND #iqUDT_WorkstationStatus."190".PEC_EoS.PEC)
	                    OR (#sx_LeftPushOutActiveStation1 AND #iqUDT_WorkstationStatus."210".PEC_EoS.PEC AND #sUDT_Interface211.ActualSpeed <> 0);

	                    #sFB_Conveyor190(iUDT_ConveyorConfiguration := #iUDT_Configuration."190".Conveyor,
	                                     idi_PECEoSDistance := #iUDT_Configuration."190".PEC_Eos.Distance,
	                                     idi_PECBoSDistance := 0,
	                                     ii_ExternalSpeed := 0,
	                                     ix_SafetyOk := #ix_SafetyOk,
	                                     ix_24vOk := #ix_24vOk,
	                                     ix_400vOk := #ix_400vOk,
	                                     ix_HardwareOk := #iUDT_HardwareOk."190",
	                                     ix_PECEoS := #iqUDT_WorkstationStatus."190".PEC_EoS.PEC,
	                                     ix_PECBoS := TRUE,
	                                     ix_ReverseDirection := FALSE,
	                                     ix_ExternalRequestDieBack := FALSE,
	                                     ix_ExternalRequestHold := #sx_LeftExternalRequestHold190,
	                                     ix_ResetEnergySave := FALSE,
	                                     qUDT_HMIStatus => #iqUDT_WorkstationStatus."190".Conveyor,
	                                     qUDT_Status => #iqUDT_WorkstationCommonStatus."190",
	                                     iqUDT_EquipmentControl := #iqUDT_EquipmentControl,
	                                     iqUDT_ConveyorCommand := #iqUDT_WorkstationCommands."190".Conveyor,
	                                     iqUDT_ConveyorInterface := #sUDT_Interface190,
	                                     iqUDT_HandShakeUp := #sUDT_Handshake180,
	                                     iqUDT_HandShake := #sUDT_Handshake190,
	                                     iqUDT_Statistics := #iqUDT_WorkstationStatistics."190".Conveyor);
	                END_REGION

	                REGION MCO

	                    #sFB_MCOConveyLinxAixController190(iUDT_AixConfig := #iUDT_Configuration."190".MCO_M01,
	                                                       iv_AixInputsModule := #iUDT_MotorInput190,
	                                                       ix_24vOk := #ix_24vOk,
	                                                       ix_SimulationModeActive := "DB_Memory".Simulation,
	                                                       ii_MotorPositionId := 1,
	                                                       qUDT_HMIStatus => #iqUDT_WorkstationStatus."190".MCO_M01,
	                                                       iqv_AixOutputsModule := #iqUDT_MotorOutput190,
	                                                       iqUDT_ConveyorInterface := #sUDT_Interface190,
	                                                       iqUDT_MCOStatistics := #iqUDT_WorkstationStatistics."190".MCO_M01);
	                END_REGION
	            END_REGION

	            REGION 210

	                REGION Displacement

	                    #sFB_Displacement210(#sUDT_Interface210);

	                END_REGION

	                REGION MCO

